Fanuc KAREL source: kb00023.KL

PROGRAM KB00023
%NOLOCKGROUP
VAR
P1:INTEGER;P2:INTEGER
BEGIN
--
P1=1
P2=1
CLOSE_TPE(P1,P2)
END KB00023
